(* IEC 61131-3 sources: test/Class/Sfc_Parallel_Handler_Base, 1 file *)

(* ---- Sfc_Parallel_Handler_Base.st ---- *)
(*!
<Class
	Name               = "Sfc_Parallel_Handler_Base"
	Revision           = "1.0"
	RealtimeTask       = "false"
	CyclicTask         = "false"
	BackgroundTask     = "false"
	Sigmatek           = "true"
	OSInterface        = "false"
	HighPriority       = "false"
	Automatic          = "false"
	UpdateMode         = "Prescan"
	SharedCommandTable = "true"
	Objectsize         = "(284,120)"
	Comment            = "Helper class for joining parallel branches.">
	<Channels>
		<Server Name="Itf" Visualized="false" Initialize="false" WriteProtected="true" Retentive="false"/>
		<Client Name="CallTransition" Required="false" Internal="false"/>
	</Channels>
</Class>
*)
Sfc_Parallel_Handler_Base : CLASS
  //Servers:
	Itf 	: SvrChCmd_DINT;
  //Clients:
	CallTransition 	: CltCh_DINT;
  //Variables:
  //Functions:

	FUNCTION VIRTUAL ReadyForTrans
		VAR_OUTPUT
			Result 	: BOOL;
		END_VAR;

	FUNCTION VIRTUAL GLOBAL Itf::Read
		VAR_OUTPUT
			output (EAX) 	: DINT;
		END_VAR;
  //Tables:
	FUNCTION @STD
		VAR_OUTPUT
			ret_code	: CONFSTATES;
		END_VAR;
	FUNCTION GLOBAL TAB @CT_;
END_CLASS;

FUNCTION VIRTUAL GLOBAL Sfc_Parallel_Handler_Base::Itf::Read
	VAR_OUTPUT
		output (EAX) 	: DINT;
	END_VAR

  output := 0;

  if ReadyForTrans() = true then

    output := CallTransition.Read();

  end_if;

END_FUNCTION

FUNCTION VIRTUAL Sfc_Parallel_Handler_Base::ReadyForTrans
	VAR_OUTPUT
		Result 	: BOOL;
	END_VAR

  Result := FALSE;

END_FUNCTION
